// TwinCAT 3 PLC project Simulator
// ProgramVersion: 3.1.4023.0
// libraries:
//   Tc2_Standard, * (Beckhoff Automation GmbH)
//   Tc2_System, * (Beckhoff Automation GmbH)
//   Tc2_Utilities, * (Beckhoff Automation GmbH)
//   Tc3_Module, * (Beckhoff Automation GmbH)
// project tree:
//   DUTs/ EachRecipeStep.TcDUT, PhysicalIO.TcDUT, Pump.TcDUT, Reactor.TcDUT, Valve.TcDUT, Vessel.TcDUT, VFD.TcDUT
//   GVLs/ IO.TcGVL, R1.TcGVL
//   Helpers/ RemainingTimeCalculator.TcPOU, ShutDown.TcPOU, Simulator.TcPOU
//   / PlcTask.TcTTO
//   POUs/ MAIN.TcPOU
//   RecipeModules/ InitializeRecipeModule.TcPOU, RecipeModule_R1.TcPOU

CONFIGURATION Simulator
    RESOURCE PLC ON TwinCAT3
        TASK PlcTask(INTERVAL := T#100000us, PRIORITY := 20);
        PROGRAM MAIN WITH PlcTask : MAIN;
    END_RESOURCE
END_CONFIGURATION

// ---- DUTs/EachRecipeStep.TcDUT
TYPE EachRecipeStep :
STRUCT

   ///Tags for start block
     HeatCoolModeSelection:BOOL:=0; /// 0-is jacket mode/ 1-is process mode
	 HeatCoolDeltaTemp:DINT:=0; 
	 Started:BOOL:=0;
	 StartedTime:STRING:='';
	 Ended:BOOL:=0;
	 EndedTime:STRING:='';

	///Tags for HeatCoolBlock
	HeatCoolEnabled:BOOL:=0;
	HeatCoolStarted:BOOL:=0;
	HeatCoolStartedTime:STRING:='';
	HeatCoolEnded:BOOL:=0;
	HeatCoolEndedTime:STRING:='';
	HeatCoolSetPointExpression:DINT:=0;
	HeatCoolDuration:DINT:=0;
	HeatCoolOperatingMode:BOOL:=0;
	
	///Tags for StirrerBlock
	StirrerEnabled:BOOL:=0;
	StirrerStarted:BOOL:=0;
	StirrerStartedTime:STRING:='';
	StirrerEnded:BOOL:=0;
	StirrerEndedTime:STRING:='';
	StirrerSetPointExpression:DINT:=0;

	///Tags for DoseBlock	
	DosingEnabled:BOOL:=0;
	DosingStarted:BOOL:=0;
	DosingStartedTime:STRING:='';
	DosingEnded:BOOL:=0;
	DosingEndedTime:STRING:='';
    DosingMaxAmount:REAL:=0;
	DosingStopTemp:DINT:=0;
	DosingResumeTemp:DINT:=0;
	DosingRateSetpointExpression:REAL:=0;
	DosingMinRate:DINT:=0;
	DosingMaxRate:DINT:=0;
	DosingSettlingTime:DINT:=0;
	DosingMinPh:DINT:=0;
	DosingMaxPh:DINT:=0;
	DosingOperatingMode:BOOL:=0;
	
	////Tags for Wait tags
	WaitEnabled:BOOL:=0;
	WaitStarted:BOOL:=0;
	WaitStartedTime:STRING:='';
	WaitEndedTime:STRING:='';
	WaitEnded:BOOL:=0;
	WaitDuration:DINT:=0;
	WaitRemainingSeconds : INT;
	WaitRemainingMinutes : INT;
	WaitRemainingTime : STRING;
	
	//Tags for Centrifuge Block
	CentrifugeEnabled : BOOL;
	CentrifugeStarted : BOOL;
	CentrifugeEnded : BOOL;
	CentrifugeSpeedSetPoint : DINT;
	CentrifugeWaitTime : DINT;
	
	//Tags for Valves Block
	ValvesEnabled : BOOL;
	ValvesStarted : BOOL;
	ValvesEnded : BOOL;
	ValveAStatus : BOOL;
	ValveBStatus : BOOL;
	ValveCStatus : BOOL;
	
	//Tags for AOOD Pump Block
	AOODPumpEnabled : BOOL;
	AOODPumpStarted : BOOL;
	AOODPumpEnded : BOOL;
	Pump1Status : BOOL;
	Pump2Status : BOOL;

END_STRUCT
END_TYPE

// ---- DUTs/PhysicalIO.TcDUT
TYPE PhysicalIO :
STRUCT
	R1_Valves AT %Q* : ARRAY[0..7] OF BOOL;
	R1_Pumps AT %Q* : ARRAY[0..1] OF BOOL;
	R1_LS AT %I* : ARRAY[0..1] OF BOOL;

	R2_Valves AT %Q* : ARRAY[0..7] OF BOOL;
	R2_Pumps AT %Q* : ARRAY[0..1] OF BOOL;
	R2_LS AT %I* : ARRAY[0..1] OF BOOL;

	R3_Valves AT %Q* : ARRAY[0..7] OF BOOL;
	R3_Pumps AT %Q* : ARRAY[0..1] OF BOOL;
	R3_LS AT %I* : ARRAY[0..1] OF BOOL;

	R4_Valves AT %Q* : ARRAY[0..7] OF BOOL;
	R4_Pumps AT %Q* : ARRAY[0..1] OF BOOL;
	R4_LS AT %I* : ARRAY[0..1] OF BOOL;

	R5_Valves AT %Q* : ARRAY[0..7] OF BOOL;
	R5_Pumps AT %Q* : ARRAY[0..1] OF BOOL;
	R5_LS AT %I* : ARRAY[0..1] OF BOOL;

	AA1_Valves AT %Q* : ARRAY[0..7] OF BOOL;
	AA1_Pumps AT %Q* : ARRAY[0..1] OF BOOL;
	AA1_LS AT %I* : ARRAY[0..1] OF BOOL;

	AA2_Valves AT %Q* : ARRAY[0..7] OF BOOL;
	AA2_Pumps AT %Q* : ARRAY[0..1] OF BOOL;
	AA2_LS AT %I* : ARRAY[0..1] OF BOOL;

	MVB_Valves AT %Q* : ARRAY[0..7] OF BOOL;
	MVB_Pumps AT %Q* : ARRAY[0..1] OF BOOL;
	MVB_LS AT %I* : ARRAY[0..1] OF BOOL;

	DCM_Valves AT %Q* : ARRAY[0..7] OF BOOL;
	DCM_Pumps AT %Q* : ARRAY[0..1] OF BOOL;
	DCM_LS AT %I* : ARRAY[0..1] OF BOOL;

	RV_Valves AT %Q* : ARRAY[0..7] OF BOOL;
	RV_Pumps AT %Q* : ARRAY[0..1] OF BOOL;
	RV_AI AT %I* : ARRAY[0..4] OF INT;
	RV_AO AT %Q* : ARRAY[0..1] OF INT;

	MVA_Valves AT %Q* : ARRAY[0..7] OF BOOL;
	MVA_Pumps AT %Q* : ARRAY[0..1] OF BOOL;
	MVA_AI AT %I* : ARRAY[0..4] OF INT;
	MVA_AO AT %Q* : ARRAY[0..1] OF INT;


END_STRUCT
END_TYPE

// ---- DUTs/Pump.TcDUT
TYPE Pump EXTENDS Valve :
STRUCT
	nPulse : INT;
	sTime : STRING;
	sRemainingTime : STRING;
END_STRUCT
END_TYPE

// ---- DUTs/Reactor.TcDUT
TYPE Reactor EXTENDS Vessel :
STRUCT
	TemperatureInputRaw : INT;
	PressureInputRaw : INT;
	LevelInputRaw : INT;
	
	VFD : VFD;
END_STRUCT
END_TYPE

// ---- DUTs/Valve.TcDUT
TYPE Valve :
STRUCT
	bStart : BOOL;
	Output : BOOL;
	
	
END_STRUCT
END_TYPE

// ---- DUTs/Vessel.TcDUT
TYPE Vessel :
STRUCT
	LLS : BOOL;	
	ULS : BOOL;	
	
	Valves : ARRAY[0..7] OF Valve;
	Pumps : ARRAY[0..1] OF Pump; 
//	VentValve : Valve;
//	N2PurgeValve : Valve;
//	TransferValve : Valve;
//	FillInValve : Valve;
//	FillInHeaderValve : Valve;
// 	DrainValve : Valve;
//	FlushingValve : Valve;

//	FillInPump : PUMP;
//	TransferPump : PUMP;
	
	
	
END_STRUCT
END_TYPE

// ---- DUTs/VFD.TcDUT
TYPE VFD :
STRUCT
	bStart : BOOL;
	bStop : BOOL;
	nRPMSetPointScaled : REAL;
	nRPMFeedBackScaled : REAL;
	nRPMFeedBackRaw : INT;
	
	nRPMSetPointRaw : INT;

	
END_STRUCT
END_TYPE

// ---- GVLs/IO.TcGVL
{attribute 'qualified_only'}
VAR_GLOBAL
	(*Recipe..5, AA1, AA2, DCM, MVB*)
	Vessels : ARRAY[0..8] OF Vessel; 
	(* MVA, RV *)
	Reactors : ARRAY[0..2] OF Reactor;
	Pressure_1 : LREAL;
	Pressure_2 : LREAL;
	PH_1 : LREAL;
	PH_2 : LREAL;
	Temperature_1 : LREAL;
	Temperature_2 : LREAL;
	StirrerCommand_1 : BOOL;
	StirrerCommand_2 : BOOL;
	StirrerSetPoint_1 : LREAL;
	StirrerSetPoint_2 : LREAL;
	
	PhysicalIO : PhysicalIO;
END_VAR

// ---- GVLs/R1.TcGVL
VAR_GLOBAL
	//***** TAGS FOR HC ******//
	HeatCoolStatus : BOOL;
	HeatCoolSetPoint : DINT := 0;
	HeatCoolTemperatureControlType : BOOL; (* 0 - Jacket , 1 - Process *)
	HeatCoolStatusFeedback : BOOL;
	ReactorMassTemperature : REAL;
	JacketOutletTemperature : REAL;
	
// ***** TAGS FOR STIRRER *****//
	StirrerStatus : BOOL;
	StirrerStatusFeedback : BOOL;
	StirrerSetPoint : DINT;
	StirrerRPM : DINT;  (* Rotations Per Minute *)
	
// ***** TAGS FOR DOSING PUMP ******//
	DosingPumpStatus : BOOL;
	DosingPumpFlowSetPoint : REAL;
	DosingPumpFPM : REAL; (* Flow Per Minute *)
	DosingPumpStatusFeedback : BOOL;
	

//***** COMPULSORY UI TAGS *****//
	UsedNow : BOOL :=FALSE;
	EmergencyStatus :BOOL:=0;
	BatchText_1:STRING;
	BatchText_2:STRING;
	BatchText_3:STRING;
	BatchText_4:STRING;
	BatchText_5:STRING;


//****** TAGS FOR RECIPE ******//
	StepCount:INT:=0;
	TotalEnabledValue:INT:=0;
	TotalEndedValue:INT:=0;
	StepCompleted:BOOL:=0;
	NumberOfRecipeSteps : DINT := 0;
	RecipeStep: ARRAY[0..100] OF EachRecipeStep;
	RecipeStatus:BOOL:=0;
	ClearRecipe:BOOL:=0;
	AbortRecipe : BOOL := 0;
	RecipeEnded:BOOL;
	StartWaitTimer: BOOL; 
	DosingControlModeEmergency : BOOL;
	WaitTick:INT:=0;
	WaitSecondTick:INT:=0;
	WaitMinuteTick:INT:=0;
	ClearRecipeTrig:BOOL;
END_VAR

// ---- POUs/MAIN.TcPOU
PROGRAM MAIN
VAR
	recipeInitializer : InitializeRecipeModule;
	fglocal : FB_LocalSystemTime;
	System_Time: TIMESTRUCT;
	currentHour : STRING;
	currentMinute : STRING;
	concatenatedHourMinuteString : STRING;
	
	ClearRecipeTrig_R1:R_Trig;
	NullRecipeStepArray : ARRAY[0..100] OF EachRecipeStep;
	
	CameraStatus : BOOL;
	LampStatus : BOOL;
	simulator : Simulator;
	random_value : REAL;
	
	timeCounter : INT;
	updateAllParameters : BOOL;
	skipCycleCounter : INT := 0;
END_VAR

IF updateAllParameters THEN
	//Update parameters for R1 using Simulator logic
	random_value := 0;
	simulator(CurrentValue := R1.JacketOutletTemperature, TargetValue := DINT_TO_REAL(R1.HeatCoolSetPoint), SimulatedValue => R1.JacketOutletTemperature);
	simulator(CurrentValue := R1.ReactorMassTemperature, TargetValue := R1.JacketOutletTemperature, SimulatedValue => R1.ReactorMassTemperature);
	
	random_value := 0;
	simulator(CurrentValue := DINT_TO_REAL(R1.StirrerRPM), TargetValue := DINT_TO_REAL(R1.StirrerSetPoint), SimulatedValue => random_value);
	R1.StirrerRPM := REAL_TO_INT(random_value);
	
	//Reset timeCounter
	updateAllParameters := FALSE;
	timeCounter := 0;
ELSE
	timeCounter := timeCounter + 1;
	IF timeCounter >= 5 THEN
		updateAllParameters := TRUE;
	END_IF
END_IF

recipeInitializer(GvlIdentifier := 1, ClearRecipe := R1.ClearRecipe);

END_PROGRAM

// ---- RecipeModules/InitializeRecipeModule.TcPOU
FUNCTION_BLOCK InitializeRecipeModule
VAR_INPUT
	GvlIdentifier : INT;
	ClearRecipe : BOOL;
END_VAR
VAR_OUTPUT
END_VAR
VAR
	NullRecipeStepArray : ARRAY[0..100] OF EachRecipeStep;
	ClearRecipeTrig:R_Trig;
END_VAR

CASE GvlIdentifier OF
	1:
		IF R1.RecipeStatus THEN
			RecipeModule_R1();
		END_IF
	  
	////End condition to wipe of the data in structure
		ClearRecipeTrig(clk:=R1.ClearRecipe,q=>);
		 IF ClearRecipeTrig.Q  THEN
			R1.RecipeStatus:=FALSE;
			R1.RecipeStep := NullRecipeStepArray;
			R1.ClearRecipe:=FALSE;
			R1.RecipeEnded:=FALSE;
			R1.StepCount:=0;
			RecipeModule_R1.DosingTotalizerVolume:=0;
		END_IF
	ELSE
		RETURN;
END_CASE

END_FUNCTION_BLOCK

// ---- RecipeModules/RecipeModule_R1.TcPOU
PROGRAM RecipeModule_R1
VAR
	shutDownFB:Shutdown;
	remainingTimeCalculator : RemainingTimeCalculator;
	temperature : DINT := 0;
	
	DosingTick: INT;
	AbortTrig:R_Trig;
END_VAR
VAR_INPUT
	DosingTotalizerVolume: REAL;
END_VAR

IF R1.RecipeStep[0].Started AND R1.RecipeStep[0].StartedTime = '' THEN
	//Update StartedTime
	R1.RecipeStep[0].StartedTime := MAIN.concatenatedHourMinuteString;
END_IF

// Start Block and HC Mode Selection
IF R1.RecipeStep[R1.StepCount].Started THEN
  R1.StepCount:= R1.StepCount+1;
 // R1.AbortRecipe:=FALSE;
  R1.ClearRecipe:=FALSE;
  R1.RecipeEnded:=FALSE;
END_IF  
 
// Check Process or JACKET SELECTION
IF R1.RecipeStep[0].HeatCoolModeSelection THEN
	R1.HeatCoolTemperatureControlType:=TRUE;
	temperature:=REAL_TO_DINT(R1.ReactorMassTemperature);
ELSE
	R1.HeatCoolTemperatureControlType:=FALSE;	
	temperature:=REAL_TO_DINT(R1.JacketOutletTemperature);
END_IF

 IF R1.RecipeStep[R1.StepCount].HeatcoolEnabled THEN
	R1.HeatCoolSetPoint:=R1.RecipeStep[R1.StepCount].HeatCoolSetpointExpression;		
	R1.RecipeStep[R1.StepCount].HeatCoolStarted :=TRUE;
	IF R1.RecipeStep[R1.StepCount].HeatCoolStartedTime = '' THEN
		R1.RecipeStep[R1.StepCount].HeatCoolStartedTime := Main.concatenatedHourMinuteString;
	END_IF
	R1.HeatCoolStatus:=TRUE;
	
		///Check for condition in step  
	 IF ABS(temperature-R1.RecipeStep[R1.StepCount].HeatCoolSetpointExpression )<0.5 THEN
		R1.RecipeStep[R1.StepCount].HeatcoolEnded :=TRUE;	
		IF R1.RecipeStep[R1.StepCount].HeatCoolEndedTime = '' THEN
			R1.RecipeStep[R1.StepCount].HeatCoolEndedTime := Main.concatenatedHourMinuteString;
		END_IF
	 END_IF     	
 END_IF
	
////Recipe block for stirrer
IF R1.RecipeStep[R1.StepCount].StirrerEnabled THEN
	R1.StirrerSetPoint:=R1.RecipeStep[R1.StepCount].StirrerSetPointExpression;
	R1.StirrerStatus:=TRUE;	
    R1.RecipeStep[R1.StepCount].StirrerStarted:=TRUE;
	IF R1.RecipeStep[R1.StepCount].StirrerStartedTime = '' THEN
		R1.RecipeStep[R1.StepCount].StirrerStartedTime := Main.concatenatedHourMinuteString;
	END_IF
	
	///Check the Actual speed to end the step
      IF ABS(R1.StirrerRPM- R1.RecipeStep[R1.StepCount].StirrerSetPointExpression)<8 THEN
		R1.RecipeStep[R1.StepCount].StirrerEnded:=TRUE;
		IF R1.RecipeStep[R1.StepCount].StirrerEndedTime = '' THEN
			R1.RecipeStep[R1.StepCount].StirrerEndedTime := Main.concatenatedHourMinuteString;
		END_IF
	  END_IF
	//Check the rpm TO switch off the vfd
	  IF R1.RecipeStep[R1.StepCount].StirrerSetPointExpression=0 THEN
		R1.StirrerStatus:=FALSE;	
	  END_IF///
  END_IF 


(*////Wait Block*)
IF R1.RecipeStep[R1.StepCount].WaitEnabled AND NOT R1.RecipeStep[StepCount].WaitEnded THEN
    R1.RecipeStep[R1.StepCount].WaitStarted:=TRUE;
	IF R1.RecipeStep[R1.StepCount].WaitStartedTime = '' THEN
		R1.RecipeStep[R1.StepCount].WaitStartedTime := Main.concatenatedHourMinuteString;
	END_IF
	R1.WaitTick:=R1.WaitTick+1;
	IF R1.WaitTick=10  THEN
		//Update the Second Tick
		R1.WaitSecondTick:=R1.WaitSecondTick+1;
		R1.WaitTick:=0;
	END_IF
		
	IF  R1.WaitSecondTick=60  THEN
		//Update the Minute Tick
		R1.WaitMinuteTick:=R1.WaitMinuteTick+1;
		R1.WaitSecondTick:=0;
	END_IF	

	//Update the Remaining Time
	remainingTimeCalculator(elapsedSeconds:= R1.WaitSecondTick, elapsedMinutes:= R1.WaitMinuteTick, givenDuration:= DINT_TO_INT(R1.RecipeStep[R1.StepCount].WaitDuration), 
							leftOverSeconds=> R1.RecipeStep[R1.StepCount].WaitRemainingSeconds, leftOverMinutes=> R1.RecipeStep[R1.StepCount].WaitRemainingMinutes);
	R1.RecipeStep[R1.StepCount].WaitRemainingTime := INT_TO_STRING(R1.RecipeStep[R1.StepCount].WaitRemainingMinutes);
	R1.RecipeStep[R1.StepCount].WaitRemainingTime := CONCAT(STR1:= R1.RecipeStep[R1.StepCount].WaitRemainingTime, STR2:= ':');
	R1.RecipeStep[R1.StepCount].WaitRemainingTime := CONCAT(STR1:= R1.RecipeStep[R1.StepCount].WaitRemainingTime, STR2:= INT_TO_STRING(R1.RecipeStep[R1.StepCount].WaitRemainingSeconds));
	
	(*///To write ended time*)
	IF ABS(R1.WaitMinuteTick -R1.RecipeStep[R1.StepCount].WaitDuration)=0 THEN
		R1.RecipeStep[R1.StepCount].WaitEnded:=TRUE;
		IF R1.RecipeStep[R1.StepCount].WaitEndedTime = '' THEN
			R1.RecipeStep[R1.StepCount].WaitEndedTime := Main.concatenatedHourMinuteString;
		END_IF
		R1.WaitTick:=0;
		R1.WaitSecondTick:=0;
		R1.WaitMinuteTick:=0;
	END_IF
END_IF
	
IF R1.RecipeStep[StepCount].DosingEnabled AND NOT R1.RecipeStep[StepCount].DosingEnded THEN
	R1.RecipeStep[StepCount].DosingStarted := TRUE;
	IF R1.RecipeStep[R1.StepCount].DosingStartedTime = '' THEN
		R1.RecipeStep[R1.StepCount].DosingStartedTime := Main.concatenatedHourMinuteString;
	END_IF
	//Update Totalized Volume
		IF  R1.DosingPumpStatus THEN
			DosingTick:=DosingTick+1;
		END_IF
		   
	  IF DosingTick=100 THEN
		  DosingTotalizerVolume:=DosingTotalizerVolume+(R1.RecipeStep[StepCount].DosingRateSetpointExpression/2.7 * 0.045);	  
	  END_IF
	  
	  IF DosingTick>100 THEN
		  DosingTick:=0;
	  END_IF
	  
	IF DosingTotalizerVolume < R1.RecipeStep[StepCount].DosingMaxAmount THEN
		IF R1.DosingPumpStatus THEN
			IF temperature < R1.RecipeStep[StepCount].DosingStopTemp THEN
				R1.DosingPumpStatus := TRUE;
				R1.DosingPumpFlowSetPoint := R1.RecipeStep[StepCount].DosingRateSetpointExpression;
			ELSE
				R1.DosingPumpStatus := FALSE;
				R1.DosingPumpFlowSetPoint := 0;
			END_IF
		ELSE
			IF DosingTotalizerVolume = 0 AND temperature > R1.RecipeStep[StepCount].DosingResumeTemp AND temperature < R1.RecipeStep[StepCount].DosingStopTemp THEN
				//Logic for starting Dosing Pump First Time in a Recipe Step
				R1.DosingPumpStatus := TRUE;
				R1.DosingPumpFlowSetPoint := R1.RecipeStep[StepCount].DosingRateSetpointExpression;
			END_IF
			
			IF temperature < R1.RecipeStep[StepCount].DosingResumeTemp THEN
				R1.DosingPumpStatus := TRUE;
				R1.DosingPumpFlowSetPoint := R1.RecipeStep[StepCount].DosingRateSetpointExpression;
			END_IF
		END_IF
	ELSE
		R1.DosingPumpStatus := FALSE;
		R1.DosingPumpFlowSetPoint := 0;
		R1.RecipeStep[StepCount].DosingEnded := TRUE;
		IF R1.RecipeStep[R1.StepCount].DosingEndedTime = '' THEN
			R1.RecipeStep[R1.StepCount].DosingEndedTime := Main.concatenatedHourMinuteString;
		END_IF
		DosingTick := 0;
		DosingTotalizerVolume:=0;
	END_IF
END_IF

IF R1.StepCount>0 THEN 

(*//Step control block To increment to next step*)
 R1.TotalEnabledValue:=BOOL_TO_INT(R1.RecipeStep[R1.StepCount].HeatcoolEnabled)+BOOL_TO_INT(R1.RecipeStep[R1.StepCount].StirrerEnabled)+BOOL_TO_INT(R1.RecipeStep[R1.StepCount].WaitEnabled)+BOOL_TO_INT( R1.RecipeStep[R1.StepCount].DosingEnabled);
 R1.TotalEndedValue:=BOOL_TO_INT(R1.RecipeStep[R1.StepCount].HeatCoolEnded)+BOOL_TO_INT(R1.RecipeStep[R1.StepCount].StirrerEnded)+BOOL_TO_INT(R1.RecipeStep[R1.StepCount].WaitEnded)+BOOL_TO_INT( R1.RecipeStep[R1.StepCount].DosingEnded);

    IF (R1.TotalEnabledValue - R1.TotalEndedValue)=0 THEN 
		R1.StepCount:=R1.StepCount+1;
    END_IF
END_IF
  
 (* ///To End the Recipe**)
 IF  R1.NumberOfRecipeSteps = R1.StepCount THEN
	 R1.StirrerStatus:=FALSE;
	 R1.StirrerSetPoint:=0;
	 R1.HeatCoolStatus:=FALSE;
	 R1.HeatCoolSetPoint:=0;	
     R1.StepCompleted:=FALSE;	 
	 R1.RecipeEnded:=TRUE;
	 R1.RecipeStatus:=FALSE;
 END_IF
  
(* //TO ABORT RECIPE*)
AbortTrig(CLK:=R1.AbortRecipe,Q=>);
IF AbortTrig.Q THEN
	shutDownFB(GvlIdentifier := 'R1');
	AbortTrig.CLK := FALSE;
END_IF

END_PROGRAM

// ---- Helpers/ShutDown.TcPOU
FUNCTION_BLOCK PUBLIC ShutDown
VAR_INPUT
	GvlIdentifier : STRING;
END_VAR
VAR_OUTPUT
END_VAR
VAR
END_VAR

IF GvlIdentifier = 'R1' THEN
	R1.RecipeStatus := FALSE;
	R1.HeatCoolStatus := FALSE;
	R1.StirrerStatus := FALSE;
	R1.AbortRecipe := FALSE;
	R1.DosingPumpStatus :=FALSE;
END_IF

END_FUNCTION_BLOCK

// ---- Helpers/RemainingTimeCalculator.TcPOU
FUNCTION_BLOCK PUBLIC RemainingTimeCalculator
VAR_INPUT
	elapsedSeconds : INT;
	elapsedMinutes : INT;
	givenDuration : INT; //Assume Duration in Minutes by default
END_VAR
VAR_OUTPUT
	leftOverSeconds : INT;
	leftOverMinutes : INT;
END_VAR
VAR
END_VAR

IF givenDuration <= elapsedMinutes THEN
	leftOverSeconds := 0;
	leftOverMinutes := 0;
ELSE
	leftOverMinutes := givenDuration - elapsedMinutes - 1;
	leftOverSeconds := 60 - elapsedSeconds;
END_IF

END_FUNCTION_BLOCK

// ---- Helpers/Simulator.TcPOU
FUNCTION_BLOCK Simulator
VAR_INPUT
	CurrentValue : REAL;
	TargetValue : REAL;
END_VAR
VAR_OUTPUT
	SimulatedValue : REAL;
END_VAR
VAR
	random_value : LREAL;
	fb_ran : DRAND;
END_VAR

fb_ran(Seed := 0, Num => random_value);
random_value := 0.5 * STRING_TO_REAL(LREAL_TO_FMTSTR(random_value, 2, TRUE));
IF ABS(CurrentValue-TargetValue)>0.5 THEN
	IF CurrentValue < TargetValue THEN
		CurrentValue := CurrentValue + random_value;
	ELSE
		CurrentValue := CurrentValue - random_value;
	END_IF
END_IF
SimulatedValue := STRING_TO_REAL(LREAL_TO_FMTSTR(CurrentValue, 2, TRUE)); //Rounding again here to clear any errors above

END_FUNCTION_BLOCK
